{attribute 'qualified_only'}
{attribute 'strict'}
TYPE EFeedbackMsgChuckBase :
(
	IsInLoadingPositionMsg := 10
);
END_TYPE

(* stored: Version 1.1.0.1, ProductVersion 3.1.4024.12
   DUT EFeedbackMsgChuckBase: Id {7059d108-cdc8-4f99-9f10-14740e977e7e} *)
